DATA_BLOCK "DB_Z256_Scada"
{ DB_Accessible_From_OPC_UA := 'FALSE' ;
 DB_Accessible_From_Webserver := 'FALSE' ;
 S7_Optimized_Access := 'FALSE' }
VERSION : 0.1
NON_RETAIN
   STRUCT
      tAlm : Struct   // HMI Alarms
         tE { ExternalWritable := 'False'} : Struct
            x0 { ExternalWritable := 'False'} : Bool;   // KE.Main emergency on
            x1 { ExternalWritable := 'False'} : Bool;   // KE1.Local emergency on
            x2 { ExternalWritable := 'False'} : Bool;   // Cabinet.Emergency localization
            x3 { ExternalWritable := 'False'} : Bool;   // SB1.Emergency localization
            x4 { ExternalWritable := 'False'} : Bool;   // SB2.Emergency localization
            x5 { ExternalAccessible := 'False'; ExternalVisible := 'False'; ExternalWritable := 'False'} : Bool;
            x6 { ExternalAccessible := 'False'; ExternalVisible := 'False'; ExternalWritable := 'False'} : Bool;
            x7 { ExternalAccessible := 'False'; ExternalVisible := 'False'; ExternalWritable := 'False'} : Bool;
            x8 { ExternalAccessible := 'False'; ExternalVisible := 'False'; ExternalWritable := 'False'} : Bool;
            x9 { ExternalAccessible := 'False'; ExternalVisible := 'False'; ExternalWritable := 'False'} : Bool;
            x10 { ExternalAccessible := 'False'; ExternalVisible := 'False'; ExternalWritable := 'False'} : Bool;
            x11 { ExternalAccessible := 'False'; ExternalVisible := 'False'; ExternalWritable := 'False'} : Bool;
            x12 { ExternalAccessible := 'False'; ExternalVisible := 'False'; ExternalWritable := 'False'} : Bool;
            x13 { ExternalAccessible := 'False'; ExternalVisible := 'False'; ExternalWritable := 'False'} : Bool;
            x14 { ExternalAccessible := 'False'; ExternalVisible := 'False'; ExternalWritable := 'False'} : Bool;
            x15 { ExternalAccessible := 'False'; ExternalVisible := 'False'; ExternalWritable := 'False'} : Bool;
            x16 { ExternalAccessible := 'False'; ExternalVisible := 'False'; ExternalWritable := 'False'} : Bool;
            x17 { ExternalAccessible := 'False'; ExternalVisible := 'False'; ExternalWritable := 'False'} : Bool;
            x18 { ExternalAccessible := 'False'; ExternalVisible := 'False'; ExternalWritable := 'False'} : Bool;
            x19 { ExternalAccessible := 'False'; ExternalVisible := 'False'; ExternalWritable := 'False'} : Bool;
            x20 { ExternalAccessible := 'False'; ExternalVisible := 'False'; ExternalWritable := 'False'} : Bool;
            x21 { ExternalAccessible := 'False'; ExternalVisible := 'False'; ExternalWritable := 'False'} : Bool;
            x22 { ExternalAccessible := 'False'; ExternalVisible := 'False'; ExternalWritable := 'False'} : Bool;
            x23 { ExternalAccessible := 'False'; ExternalVisible := 'False'; ExternalWritable := 'False'} : Bool;
            x24 { ExternalAccessible := 'False'; ExternalVisible := 'False'; ExternalWritable := 'False'} : Bool;
            x25 { ExternalAccessible := 'False'; ExternalVisible := 'False'; ExternalWritable := 'False'} : Bool;
            x26 { ExternalAccessible := 'False'; ExternalVisible := 'False'; ExternalWritable := 'False'} : Bool;
            x27 { ExternalAccessible := 'False'; ExternalVisible := 'False'; ExternalWritable := 'False'} : Bool;
            x28 { ExternalAccessible := 'False'; ExternalVisible := 'False'; ExternalWritable := 'False'} : Bool;
            x29 { ExternalAccessible := 'False'; ExternalVisible := 'False'; ExternalWritable := 'False'} : Bool;
            x30 { ExternalAccessible := 'False'; ExternalVisible := 'False'; ExternalWritable := 'False'} : Bool;
            x31 { ExternalAccessible := 'False'; ExternalVisible := 'False'; ExternalWritable := 'False'} : Bool;
         END_STRUCT;
         tS { ExternalWritable := 'False'} : Struct
            tS0 { ExternalWritable := 'False'} : Struct
               x0 { ExternalWritable := 'False'} : Bool;   // xB18-3L+.PowerSupplyInputControlCabinetON
               x1 { ExternalWritable := 'False'} : Bool;   // xB18-7L+.InputInstallationPowerSupplyON"
               x2 { ExternalWritable := 'False'} : Bool;   // xB11QF1/1D/QF2.Anomaly power supplies 120V
               x3 { ExternalWritable := 'False'} : Bool;   // xB18QF2.Power supply 24V logic
               x4 { ExternalWritable := 'False'} : Bool;   // xB18QF3.Power supply 24V logic
               x5 { ExternalWritable := 'False'} : Bool;   // xB20QF2.Power supply 24V logic
               x6 { ExternalWritable := 'False'} : Bool;   // xB20QF3.Power supply 24V logic
               x7 { ExternalWritable := 'False'} : Bool;   // xB21QF1.Power supply 24V logic
               x8 { ExternalWritable := 'False'} : Bool;   // xB41QF1.ProtectionPowerSupplyMotorsYcut 1-4
               x9 { ExternalWritable := 'False'} : Bool;   // xB41QF2.Protection power supply 36V motors longitudinal cutting 1-4
               x10 { ExternalWritable := 'False'} : Bool;   // xB42QF1.ProtectionPowerSupplyMotorsYcut 5-8
               x11 { ExternalWritable := 'False'} : Bool;   // xB42QF2.Protection power supply 36V motors longitudinal cutting 5-8
               x12 { ExternalWritable := 'False'} : Bool;
               x13 { ExternalWritable := 'False'} : Bool;
               x14 { ExternalWritable := 'False'} : Bool;
               x15 { ExternalWritable := 'False'} : Bool;
               x16 { ExternalWritable := 'False'} : Bool;   // PLCA.Timeout receiving consumed message
               x17 { ExternalWritable := 'False'} : Bool;   // PLCB.Timeout receiving consumed message
               x18 { ExternalWritable := 'False'} : Bool;   // PLCA.Mission packet lost
               x19 { ExternalWritable := 'False'} : Bool;   // PLCB.Mission packet lost
               x20 { ExternalWritable := 'False'} : Bool;   // PLCA.Syncro packet lost
               x21 { ExternalWritable := 'False'} : Bool;   // PLCB.Syncro packet lost
               x22 { ExternalWritable := 'False'} : Bool;   // Syncro.YCut meter gap outside the limits
               x23 { ExternalWritable := 'False'} : Bool;   // Syncro.Main line meter gap outside the limits
               x24 { ExternalWritable := 'False'} : Bool;   // Syncro.Timeout receiving meter signal from main line
               x25 { ExternalWritable := 'False'} : Bool;   // Syncro.Timeout receiving syncro value from mainline
               x26 { ExternalWritable := 'False'} : Bool;   // Syncro.Unexpected syncro pulse
               x27 { ExternalWritable := 'False'} : Bool;   // Syncro.Unexpected syncro message
               x28 { ExternalWritable := 'False'} : Bool;   // Syncro.Machine not syncronized
               x29 { ExternalWritable := 'False'} : Bool;
               x30 { ExternalWritable := 'False'} : Bool;
               x31 { ExternalWritable := 'False'} : Bool;
            END_STRUCT;
            tS1 { ExternalWritable := 'False'} : Struct
               x0 { ExternalWritable := 'False'} : Bool;
               x1 { ExternalWritable := 'False'} : Bool;
               x2 { ExternalWritable := 'False'} : Bool;
               x3 { ExternalWritable := 'False'} : Bool;
               x4 { ExternalWritable := 'False'} : Bool;
               x5 { ExternalWritable := 'False'} : Bool;
               x6 { ExternalWritable := 'False'} : Bool;
               x7 { ExternalWritable := 'False'} : Bool;
               x8 { ExternalWritable := 'False'} : Bool;
               x9 { ExternalWritable := 'False'} : Bool;
               x10 { ExternalWritable := 'False'} : Bool;
               x11 { ExternalWritable := 'False'} : Bool;
               x12 { ExternalWritable := 'False'} : Bool;
               x13 { ExternalWritable := 'False'} : Bool;
               x14 { ExternalWritable := 'False'} : Bool;
               x15 { ExternalWritable := 'False'} : Bool;
               x16 { ExternalWritable := 'False'} : Bool;
               x17 { ExternalWritable := 'False'} : Bool;
               x18 { ExternalWritable := 'False'} : Bool;
               x19 { ExternalWritable := 'False'} : Bool;
               x20 { ExternalWritable := 'False'} : Bool;
               x21 { ExternalWritable := 'False'} : Bool;
               x22 { ExternalWritable := 'False'} : Bool;
               x23 { ExternalWritable := 'False'} : Bool;
               x24 { ExternalWritable := 'False'} : Bool;
               x25 { ExternalWritable := 'False'} : Bool;
               x26 { ExternalWritable := 'False'} : Bool;
               x27 { ExternalWritable := 'False'} : Bool;
               x28 { ExternalWritable := 'False'} : Bool;
               x29 { ExternalWritable := 'False'} : Bool;
               x30 { ExternalWritable := 'False'} : Bool;
               x31 { ExternalWritable := 'False'} : Bool;
            END_STRUCT;
            tS2 { ExternalWritable := 'False'} : Struct
               x0 { ExternalWritable := 'False'} : Bool;
               x1 { ExternalWritable := 'False'} : Bool;
               x2 { ExternalWritable := 'False'} : Bool;
               x3 { ExternalWritable := 'False'} : Bool;
               x4 { ExternalWritable := 'False'} : Bool;
               x5 { ExternalWritable := 'False'} : Bool;
               x6 { ExternalWritable := 'False'} : Bool;
               x7 { ExternalWritable := 'False'} : Bool;
               x8 { ExternalWritable := 'False'} : Bool;
               x9 { ExternalWritable := 'False'} : Bool;
               x10 { ExternalWritable := 'False'} : Bool;
               x11 { ExternalWritable := 'False'} : Bool;
               x12 { ExternalWritable := 'False'} : Bool;
               x13 { ExternalWritable := 'False'} : Bool;
               x14 { ExternalWritable := 'False'} : Bool;
               x15 { ExternalWritable := 'False'} : Bool;
               x16 { ExternalWritable := 'False'} : Bool;
               x17 { ExternalWritable := 'False'} : Bool;
               x18 { ExternalWritable := 'False'} : Bool;
               x19 { ExternalWritable := 'False'} : Bool;
               x20 { ExternalWritable := 'False'} : Bool;
               x21 { ExternalWritable := 'False'} : Bool;
               x22 { ExternalWritable := 'False'} : Bool;
               x23 { ExternalWritable := 'False'} : Bool;
               x24 { ExternalWritable := 'False'} : Bool;
               x25 { ExternalWritable := 'False'} : Bool;
               x26 { ExternalWritable := 'False'} : Bool;
               x27 { ExternalWritable := 'False'} : Bool;
               x28 { ExternalWritable := 'False'} : Bool;
               x29 { ExternalWritable := 'False'} : Bool;
               x30 { ExternalWritable := 'False'} : Bool;
               x31 { ExternalWritable := 'False'} : Bool;
            END_STRUCT;
            tS3 { ExternalWritable := 'False'} : Struct
               x0 { ExternalWritable := 'False'} : Bool;
               x1 { ExternalWritable := 'False'} : Bool;
               x2 { ExternalWritable := 'False'} : Bool;
               x3 { ExternalWritable := 'False'} : Bool;
               x4 { ExternalWritable := 'False'} : Bool;
               x5 { ExternalWritable := 'False'} : Bool;
               x6 { ExternalWritable := 'False'} : Bool;
               x7 { ExternalWritable := 'False'} : Bool;
               x8 { ExternalWritable := 'False'} : Bool;
               x9 { ExternalWritable := 'False'} : Bool;
               x10 { ExternalWritable := 'False'} : Bool;
               x11 { ExternalWritable := 'False'} : Bool;
               x12 { ExternalWritable := 'False'} : Bool;
               x13 { ExternalWritable := 'False'} : Bool;
               x14 { ExternalWritable := 'False'} : Bool;
               x15 { ExternalWritable := 'False'} : Bool;
               x16 { ExternalWritable := 'False'} : Bool;
               x17 { ExternalWritable := 'False'} : Bool;
               x18 { ExternalWritable := 'False'} : Bool;
               x19 { ExternalWritable := 'False'} : Bool;
               x20 { ExternalWritable := 'False'} : Bool;
               x21 { ExternalWritable := 'False'} : Bool;
               x22 { ExternalWritable := 'False'} : Bool;
               x23 { ExternalWritable := 'False'} : Bool;
               x24 { ExternalWritable := 'False'} : Bool;
               x25 { ExternalWritable := 'False'} : Bool;
               x26 { ExternalWritable := 'False'} : Bool;
               x27 { ExternalWritable := 'False'} : Bool;
               x28 { ExternalWritable := 'False'} : Bool;
               x29 { ExternalWritable := 'False'} : Bool;
               x30 { ExternalWritable := 'False'} : Bool;
               x31 { ExternalWritable := 'False'} : Bool;
            END_STRUCT;
         END_STRUCT;
         tF { ExternalAccessible := 'False'; ExternalVisible := 'False'; ExternalWritable := 'False'} : Struct
            x0 { ExternalAccessible := 'False'; ExternalVisible := 'False'; ExternalWritable := 'False'} : Bool;
            x1 { ExternalAccessible := 'False'; ExternalVisible := 'False'; ExternalWritable := 'False'} : Bool;
            x2 { ExternalAccessible := 'False'; ExternalVisible := 'False'; ExternalWritable := 'False'} : Bool;
            x3 { ExternalAccessible := 'False'; ExternalVisible := 'False'; ExternalWritable := 'False'} : Bool;
            x4 { ExternalAccessible := 'False'; ExternalVisible := 'False'; ExternalWritable := 'False'} : Bool;
            x5 { ExternalAccessible := 'False'; ExternalVisible := 'False'; ExternalWritable := 'False'} : Bool;
            x6 { ExternalAccessible := 'False'; ExternalVisible := 'False'; ExternalWritable := 'False'} : Bool;
            x7 { ExternalAccessible := 'False'; ExternalVisible := 'False'; ExternalWritable := 'False'} : Bool;
            x8 { ExternalAccessible := 'False'; ExternalVisible := 'False'; ExternalWritable := 'False'} : Bool;
            x9 { ExternalAccessible := 'False'; ExternalVisible := 'False'; ExternalWritable := 'False'} : Bool;
            x10 { ExternalAccessible := 'False'; ExternalVisible := 'False'; ExternalWritable := 'False'} : Bool;
            x11 { ExternalAccessible := 'False'; ExternalVisible := 'False'; ExternalWritable := 'False'} : Bool;
            x12 { ExternalAccessible := 'False'; ExternalVisible := 'False'; ExternalWritable := 'False'} : Bool;
            x13 { ExternalAccessible := 'False'; ExternalVisible := 'False'; ExternalWritable := 'False'} : Bool;
            x14 { ExternalAccessible := 'False'; ExternalVisible := 'False'; ExternalWritable := 'False'} : Bool;
            x15 { ExternalAccessible := 'False'; ExternalVisible := 'False'; ExternalWritable := 'False'} : Bool;
            x16 { ExternalAccessible := 'False'; ExternalVisible := 'False'; ExternalWritable := 'False'} : Bool;
            x17 { ExternalAccessible := 'False'; ExternalVisible := 'False'; ExternalWritable := 'False'} : Bool;
            x18 { ExternalAccessible := 'False'; ExternalVisible := 'False'; ExternalWritable := 'False'} : Bool;
            x19 { ExternalAccessible := 'False'; ExternalVisible := 'False'; ExternalWritable := 'False'} : Bool;
            x20 { ExternalAccessible := 'False'; ExternalVisible := 'False'; ExternalWritable := 'False'} : Bool;
            x21 { ExternalAccessible := 'False'; ExternalVisible := 'False'; ExternalWritable := 'False'} : Bool;
            x22 { ExternalAccessible := 'False'; ExternalVisible := 'False'; ExternalWritable := 'False'} : Bool;
            x23 { ExternalAccessible := 'False'; ExternalVisible := 'False'; ExternalWritable := 'False'} : Bool;
            x24 { ExternalAccessible := 'False'; ExternalVisible := 'False'; ExternalWritable := 'False'} : Bool;
            x25 { ExternalAccessible := 'False'; ExternalVisible := 'False'; ExternalWritable := 'False'} : Bool;
            x26 { ExternalAccessible := 'False'; ExternalVisible := 'False'; ExternalWritable := 'False'} : Bool;
            x27 { ExternalAccessible := 'False'; ExternalVisible := 'False'; ExternalWritable := 'False'} : Bool;
            x28 { ExternalAccessible := 'False'; ExternalVisible := 'False'; ExternalWritable := 'False'} : Bool;
            x29 { ExternalAccessible := 'False'; ExternalVisible := 'False'; ExternalWritable := 'False'} : Bool;
            x30 { ExternalAccessible := 'False'; ExternalVisible := 'False'; ExternalWritable := 'False'} : Bool;
            x31 { ExternalAccessible := 'False'; ExternalVisible := 'False'; ExternalWritable := 'False'} : Bool;
         END_STRUCT;
         tW { ExternalWritable := 'False'} : Struct
            x0 { ExternalWritable := 'False'} : Bool;   // PLCA.Timeout receiving consumed message
            x1 { ExternalWritable := 'False'} : Bool;   // PLCB.Timeout receiving consumed message
            x2 { ExternalWritable := 'False'} : Bool;   // PLCA.Mission packet lost
            x3 { ExternalWritable := 'False'} : Bool;   // PLCB.Mission packet lost
            x4 { ExternalWritable := 'False'} : Bool;   // PLCA.Syncro packet lost
            x5 { ExternalWritable := 'False'} : Bool;   // PLCB.Syncro packet lost
            x6 { ExternalWritable := 'False'} : Bool;   // QF.Protection air conditioners
            x7 { ExternalAccessible := 'False'; ExternalVisible := 'False'; ExternalWritable := 'False'} : Bool;
            x8 { ExternalAccessible := 'False'; ExternalVisible := 'False'; ExternalWritable := 'False'} : Bool;
            x9 { ExternalAccessible := 'False'; ExternalVisible := 'False'; ExternalWritable := 'False'} : Bool;
            x10 { ExternalAccessible := 'False'; ExternalVisible := 'False'; ExternalWritable := 'False'} : Bool;
            x11 { ExternalAccessible := 'False'; ExternalVisible := 'False'; ExternalWritable := 'False'} : Bool;
            x12 { ExternalAccessible := 'False'; ExternalVisible := 'False'; ExternalWritable := 'False'} : Bool;
            x13 { ExternalAccessible := 'False'; ExternalVisible := 'False'; ExternalWritable := 'False'} : Bool;
            x14 { ExternalAccessible := 'False'; ExternalVisible := 'False'; ExternalWritable := 'False'} : Bool;
            x15 { ExternalAccessible := 'False'; ExternalVisible := 'False'; ExternalWritable := 'False'} : Bool;
            x16 { ExternalAccessible := 'False'; ExternalVisible := 'False'; ExternalWritable := 'False'} : Bool;
            x17 { ExternalAccessible := 'False'; ExternalVisible := 'False'; ExternalWritable := 'False'} : Bool;
            x18 { ExternalAccessible := 'False'; ExternalVisible := 'False'; ExternalWritable := 'False'} : Bool;
            x19 { ExternalAccessible := 'False'; ExternalVisible := 'False'; ExternalWritable := 'False'} : Bool;
            x20 { ExternalAccessible := 'False'; ExternalVisible := 'False'; ExternalWritable := 'False'} : Bool;
            x21 { ExternalAccessible := 'False'; ExternalVisible := 'False'; ExternalWritable := 'False'} : Bool;
            x22 { ExternalAccessible := 'False'; ExternalVisible := 'False'; ExternalWritable := 'False'} : Bool;
            x23 { ExternalAccessible := 'False'; ExternalVisible := 'False'; ExternalWritable := 'False'} : Bool;
            x24 { ExternalAccessible := 'False'; ExternalVisible := 'False'; ExternalWritable := 'False'} : Bool;
            x25 { ExternalAccessible := 'False'; ExternalVisible := 'False'; ExternalWritable := 'False'} : Bool;
            x26 { ExternalAccessible := 'False'; ExternalVisible := 'False'; ExternalWritable := 'False'} : Bool;
            x27 { ExternalAccessible := 'False'; ExternalVisible := 'False'; ExternalWritable := 'False'} : Bool;
            x28 { ExternalAccessible := 'False'; ExternalVisible := 'False'; ExternalWritable := 'False'} : Bool;
            x29 { ExternalAccessible := 'False'; ExternalVisible := 'False'; ExternalWritable := 'False'} : Bool;
            x30 { ExternalAccessible := 'False'; ExternalVisible := 'False'; ExternalWritable := 'False'} : Bool;
            x31 { ExternalAccessible := 'False'; ExternalVisible := 'False'; ExternalWritable := 'False'} : Bool;
         END_STRUCT;
      END_STRUCT;
      tHMR { ExternalWritable := 'False'} : Struct   // HMI Read
         xCalibrationsAllowed { ExternalWritable := 'False'} : Bool;   // Calibration function allowed {x|x|x|x|O}
         xSpare1 { ExternalWritable := 'False'} : Bool;
         xSpare2 { ExternalWritable := 'False'} : Bool;
         xSpare3 { ExternalWritable := 'False'} : Bool;
         xSpare4 { ExternalWritable := 'False'} : Bool;
         xSpare5 { ExternalWritable := 'False'} : Bool;
         xSpare6 { ExternalWritable := 'False'} : Bool;
         xSpare7 { ExternalWritable := 'False'} : Bool;
         xSpare8 { ExternalWritable := 'False'} : Bool;
         xSpare9 { ExternalWritable := 'False'} : Bool;
         xSpare10 { ExternalWritable := 'False'} : Bool;
         xSpare11 { ExternalWritable := 'False'} : Bool;
         xSpare12 { ExternalWritable := 'False'} : Bool;
         xSpare13 { ExternalWritable := 'False'} : Bool;
         xSpare14 { ExternalWritable := 'False'} : Bool;
         xZoneAlarm { ExternalWritable := 'False'} : Bool;   // Zone alarm {X|X|X|X|O}
         xSpare16 { ExternalWritable := 'False'} : Bool;
         xSpare17 { ExternalWritable := 'False'} : Bool;
         xSpare18 { ExternalWritable := 'False'} : Bool;
         xSpare19 { ExternalWritable := 'False'} : Bool;
         xSpare20 { ExternalWritable := 'False'} : Bool;
         xSpare21 { ExternalWritable := 'False'} : Bool;
         xSpare22 { ExternalWritable := 'False'} : Bool;
         xSpare23 { ExternalWritable := 'False'} : Bool;
         xSpare24 { ExternalWritable := 'False'} : Bool;
         xSpare25 { ExternalWritable := 'False'} : Bool;
         xSpare26 { ExternalWritable := 'False'} : Bool;
         xSpare27 { ExternalWritable := 'False'} : Bool;
         xSpare28 { ExternalWritable := 'False'} : Bool;
         xSpare29 { ExternalWritable := 'False'} : Bool;
         xSpare30 { ExternalWritable := 'False'} : Bool;
         xSpare31 { ExternalWritable := 'False'} : Bool;
         xSpare { ExternalWritable := 'False'} : Array[0..15] of Bool;
         iSpare0 { ExternalWritable := 'False'} : Int;
         iSpare1 { ExternalWritable := 'False'} : Int;
         iSpare2 { ExternalWritable := 'False'} : Int;
         iSpare3 { ExternalWritable := 'False'} : Int;
         iSpare4 { ExternalWritable := 'False'} : Int;
         iSpare5 { ExternalWritable := 'False'} : Int;
         iSpare6 { ExternalWritable := 'False'} : Int;
         iSpare7 { ExternalWritable := 'False'} : Int;
         iSpare8 { ExternalWritable := 'False'} : Int;
         iSpare9 { ExternalWritable := 'False'} : Int;
         iSpare10 { ExternalWritable := 'False'} : Int;
         iSpare11 { ExternalWritable := 'False'} : Int;
         iSpare12 { ExternalWritable := 'False'} : Int;
         iSpare13 { ExternalWritable := 'False'} : Int;
         iSpare14 { ExternalWritable := 'False'} : Int;
         iSpare15 { ExternalWritable := 'False'} : Int;
         iSpare16 { ExternalWritable := 'False'} : Int;
         dZoneMode { ExternalWritable := 'False'} : DInt;   // Zone modality (1=Manual;4=Automatic;8=Manual request) {x|x|x|x|O}
         dZoneState { ExternalWritable := 'False'} : DInt;   // Zone status (1=CycleON 2=StopCyc 4=CycleReq 8=StopReq 1024=E-Stop) {X|X|X|X|O}
         dCabinetStatusMCC { ExternalWritable := 'False'} : DInt;   // Cabinet status MCC1256B (1=OK;2=General power alarm;3=Local power alarm) {X|X|X|X|O}
         dProdModeRequest { ExternalWritable := 'False'} : DInt;   // Production modality request (1=Out of Production 3= In production) {x|x|x|x|O}
         dProdModeActual { ExternalWritable := 'False'} : DInt;   // Production modality actual (1=Out of production 3=In production 8=Out of production request 9=In production request) {x|x|x|x|O}
         dSpare5 { ExternalWritable := 'False'} : DInt;
         "rgdHeadsActualStatus[0]" { ExternalWritable := 'False'} : DInt;   // Head #1 prod. status (1=Out of production 3=In production 8=Out of production request 9=In production request) {x|x|x|x|O}
         "rgdHeadsActualStatus[1]" { ExternalWritable := 'False'} : DInt;   // Head #2 prod. status (1=Out of production 3=In production 8=Out of production request 9=In production request) {x|x|x|x|O}
         "rgdHeadsActualStatus[2]" { ExternalWritable := 'False'} : DInt;   // Head #3 prod. status (1=Out of production 3=In production 8=Out of production request 9=In production request) {x|x|x|x|O}
         "rgdHeadsActualStatus[3]" { ExternalWritable := 'False'} : DInt;   // Head #4 prod. status (1=Out of production 3=In production 8=Out of production request 9=In production request) {x|x|x|x|O}
         "rgdHeadsActualStatus[4]" { ExternalWritable := 'False'} : DInt;   // Head #5 prod. status (1=Out of production 3=In production 8=Out of production request 9=In production request) {x|x|x|x|O}
         "rgdHeadsActualStatus[5]" { ExternalWritable := 'False'} : DInt;   // Head #6 prod. status (1=Out of production 3=In production 8=Out of production request 9=In production request) {x|x|x|x|O}
         "rgdHeadsActualStatus[6]" { ExternalWritable := 'False'} : DInt;   // Head #7 prod. status (1=Out of production 3=In production 8=Out of production request 9=In production request) {x|x|x|x|O}
         "rgdHeadsActualStatus[7]" { ExternalWritable := 'False'} : DInt;   // Head #8 prod. status (1=Out of production 3=In production 8=Out of production request 9=In production request) {x|x|x|x|O}
         dSpare14 { ExternalWritable := 'False'} : DInt;
         dSpare15 { ExternalWritable := 'False'} : DInt;
         dSpare { ExternalWritable := 'False'} : Array[0..15] of DInt;
         rSpare0 { ExternalWritable := 'False'} : Real;
         rSpare1 { ExternalWritable := 'False'} : Real;
         rSpare2 { ExternalWritable := 'False'} : Real;
         rSpare3 { ExternalWritable := 'False'} : Real;
         rSpare4 { ExternalWritable := 'False'} : Real;
         rSpare5 { ExternalWritable := 'False'} : Real;
         rSpare6 { ExternalWritable := 'False'} : Real;
         rSpare7 { ExternalWritable := 'False'} : Real;
         rSpare8 { ExternalWritable := 'False'} : Real;
         tManCmd { ExternalWritable := 'False'} : Struct
            xSpare0 { ExternalWritable := 'False'} : Bool;
            xSpare1 { ExternalWritable := 'False'} : Bool;
            xSpare2 { ExternalWritable := 'False'} : Bool;
            xSpare3 { ExternalWritable := 'False'} : Bool;
            xSpare4 { ExternalWritable := 'False'} : Bool;
            xSpare5 { ExternalWritable := 'False'} : Bool;
            xSpare6 { ExternalWritable := 'False'} : Bool;
            xSpare7 { ExternalWritable := 'False'} : Bool;
            xSpare8 { ExternalWritable := 'False'} : Bool;
            xSpare9 { ExternalWritable := 'False'} : Bool;
            xSpare10 { ExternalWritable := 'False'} : Bool;
            xSpare11 { ExternalWritable := 'False'} : Bool;
            xSpare12 { ExternalWritable := 'False'} : Bool;
            xSpare13 { ExternalWritable := 'False'} : Bool;
            xSpare14 { ExternalWritable := 'False'} : Bool;
            xSpare15 { ExternalWritable := 'False'} : Bool;
            xSpare { ExternalWritable := 'False'} : Array[0..15] of Bool;
         END_STRUCT;
      END_STRUCT;
      tHMW : Struct   // HMI Write
         xAutoModeReq : Bool;   // Automatic mode request {x|x|x|x|O}
         xManModeReq : Bool;   // Manual mode request {x|x|x|x|O}
         xOutOfProdReq : Bool;   // Bridge out of production request {x|x|x|x|O}
         xInProdReq : Bool;   // Bridge in production request {x|x|x|x|O}
         xCutOnBreakEnabled { ExternalWritable := 'False'} : Bool;   // Cut during glass break {x|x|x|x|O}
         xMotorsAndCardsInitialize : Bool;   // Motors and cards initialize {x|x|x|x|M}
         xForceHeadsHoming : Bool;   // Force the homing of the heads {x|x|x|x|M}
         xPositionCalibrationRequest : Bool;   // Position calibration request {x|x|x|x|M}
         xBridgeOffsetCalibrationRequest : Bool;   // Bridge offset calibration request {x|x|x|x|M}
         xSpare9 { ExternalWritable := 'False'} : Bool;   //
         xSpare10 : Bool;   //
         xSpare11 : Bool;   //
         xSpare12 : Bool;
         xSpare13 : Bool;
         xGeneralReset : Bool;   // General reset {X|X|X|X|M}
         xFaultsReset : Bool;   // Reset faults {X|X|X|X|O}
         xHeadEnabled_1 { ExternalWritable := 'False'} : Bool;   // Head #1 enabled/disabled {x|x|x|x|O}
         xHeadEnabled_2 { ExternalWritable := 'False'} : Bool;   // Head #2 enabled/disabled {x|x|x|x|O}
         xHeadEnabled_3 { ExternalWritable := 'False'} : Bool;   // Head #3 enabled/disabled {x|x|x|x|O}
         xHeadEnabled_4 { ExternalWritable := 'False'} : Bool;   // Head #4 enabled/disabled {x|x|x|x|O}
         xHeadEnabled_5 { ExternalWritable := 'False'} : Bool;   // Head #5 enabled/disabled {x|x|x|x|O}
         xHeadEnabled_6 { ExternalWritable := 'False'} : Bool;   // Head #6 enabled/disabled {x|x|x|x|O}
         xHeadEnabled_7 { ExternalWritable := 'False'} : Bool;   // Head #7 enabled/disabled {x|x|x|x|O}
         xHeadEnabled_8 { ExternalWritable := 'False'} : Bool;   // Head #8 enabled/disabled {x|x|x|x|O}
         xSpare24 : Bool;
         xSpare25 : Bool;
         xSpare26 : Bool;
         xSpare27 : Bool;
         xSpare28 : Bool;
         xSpare29 : Bool;
         xSpare30 : Bool;
         xSpare31 : Bool;
         xSpare : Array[0..15] of Bool;
         iSpare0 : Int;
         iSpare1 : Int;
         iSpare2 : Int;
         iSpare3 : Int;
         iSpare4 : Int;
         iSpare5 : Int;
         iSpare6 : Int;
         iSpare7 : Int;
         iSpare8 : Int;
         iSpare9 : Int;
         iSpare10 : Int;
         iSpare11 : Int;
         iSpare12 : Int;
         iSpare13 : Int;
         iSpare14 : Int;
         iSpare15 : Int;
         iSpare16 : Int;
         dNumberOfLites : DInt;   // Calibration. number of lite on calibration {x|x|1|8|M}
         dMoveBridgeOffset_cmm : DInt;   // Calibration. Move all the heads of this offset {mm/100|mm|-100|100|M}
         dPressureScalerOnSample_perc : DInt;   // Pressure scaler during sample plate [%] {%|%|0|100|O}
         dSpare3 : DInt;
         dSpare4 : DInt;
         dSpare5 : DInt;
         dSpare6 : DInt;
         dSpare7 : DInt;
         dHead_Selected_1 : DInt;   // Calibration. head number selected Cut1 {x|x|1|11|M}
         dHead_Selected_2 : DInt;   // Calibration. head number selected Cut2 {x|x|1|11|M}
         dHead_Selected_3 : DInt;   // Calibration. head number selected Cut3{x|x|1|11|M}
         dHead_Selected_4 : DInt;   // Calibration. head number selected Cut4{x|x|1|11|M}
         dHead_Selected_5 : DInt;   // Calibration. head number selected Cut5{x|x|1|11|M}
         dHead_Selected_6 : DInt;   // Calibration. head number selected Cut6{x|x|1|11|M}
         dHead_Selected_7 : DInt;   // Calibration. head number selected Cut7{x|x|1|11|M}
         dHead_Selected_8 : DInt;   // Calibration. head number selected Cut8{x|x|1|11|M}
         dCutWidthTeo_cmm_1 : DInt;   // Calibration. cut width Lite 1 theorical [mm/100] {mm/100|mm|200|4000|M}
         dCutWidthTeo_cmm_2 : DInt;   // Calibration. cut width Lite 2 theorical [mm/100] {mm/100|mm|200|4000|M}
         dCutWidthTeo_cmm_3 : DInt;   // Calibration. cut width Lite 3 theorical [mm/100] {mm/100|mm|200|4000|M}
         dCutWidthTeo_cmm_4 : DInt;   // Calibration. cut width Lite 4 theorical [mm/100] {mm/100|mm|200|4000|M}
         dCutWidthTeo_cmm_5 : DInt;   // Calibration. cut width Lite 5 theorical [mm/100] {mm/100|mm|200|4000|M}
         dCutWidthTeo_cmm_6 : DInt;   // Calibration. cut width Lite 6 theorical [mm/100] {mm/100|mm|200|4000|M}
         dCutWidthTeo_cmm_7 : DInt;   // Calibration. cut width Lite 7 theorical [mm/100] {mm/100|mm|200|4000|M}
         dCutWidthTeo_cmm_8 : DInt;   // Calibration. cut width Lite 8 theorical [mm/100] {mm/100|mm|200|4000|M}
         dCutWidthReal_cmm_1 : DInt;   // Calibration. cut width Lite 1 real [mm/100] {mm/100|mm|200|4000|M}
         dCutWidthReal_cmm_2 : DInt;   // Calibration. cut width Lite 2 real [mm/100] {mm/100|mm|200|4000|M}
         dCutWidthReal_cmm_3 : DInt;   // Calibration. cut width Lite 3 real [mm/100] {mm/100|mm|200|4000|M}
         dCutWidthReal_cmm_4 : DInt;   // Calibration. cut width Lite 4 real [mm/100] {mm/100|mm|200|4000|M}
         dCutWidthReal_cmm_5 : DInt;   // Calibration. cut width Lite 5 real [mm/100] {mm/100|mm|200|4000|M}
         dCutWidthReal_cmm_6 : DInt;   // Calibration. cut width Lite 6 real [mm/100] {mm/100|mm|200|4000|M}
         dCutWidthReal_cmm_7 : DInt;   // Calibration. cut width Lite 7 real [mm/100] {mm/100|mm|200|4000|M}
         dCutWidthReal_cmm_8 : DInt;   // Calibration. cut width Lite 8 real [mm/100] {mm/100|mm|200|4000|M}
         dSpare32 : DInt;
         dSpare33 : DInt;
         dSpare34 : DInt;
         dSpare35 : DInt;
         dSpare36 : DInt;
         dSpare37 : DInt;
         dSpare38 : DInt;
         dSpare39 : DInt;
         dSpare { ExternalWritable := 'False'} : Array[0..19] of DInt;
         rSpare0 : Real;
         rSpare1 : Real;
         rSpare2 : Real;
         rSpare3 : Real;
         rSpare4 : Real;
         rSpare5 : Real;
         rSpare6 : Real;
         rSpare7 : Real;
         rSpare8 : Real;
         tManCmd : Struct
            xBrakeEngage : Bool;   // Brake engage all heads {x|x|x|x|O}
            xBrakeRelease : Bool;   // Brake release all heads {x|x|x|x|O}
            xSpare2 { ExternalWritable := 'False'} : Bool;
            xSpare3 { ExternalWritable := 'False'} : Bool;
            xSpare4 { ExternalWritable := 'False'} : Bool;
            xSpare5 { ExternalWritable := 'False'} : Bool;
            xSpare6 { ExternalWritable := 'False'} : Bool;
            xSpare7 { ExternalWritable := 'False'} : Bool;
            xSpare8 { ExternalWritable := 'False'} : Bool;
            xSpare9 { ExternalWritable := 'False'} : Bool;
            xSpare10 { ExternalWritable := 'False'} : Bool;
            xSpare11 { ExternalWritable := 'False'} : Bool;
            xSpare12 { ExternalWritable := 'False'} : Bool;
            xSpare13 { ExternalWritable := 'False'} : Bool;
            xSpare14 { ExternalWritable := 'False'} : Bool;
            xSpare15 { ExternalWritable := 'False'} : Bool;
            xSpare16 : Bool;
            xSpare17 : Bool;
            xSpare18 : Bool;
            xSpare19 : Bool;
            xSpare20 : Bool;
            xSpare21 : Bool;
            xSpare22 : Bool;
            xSpare23 : Bool;
            xSpare24 : Bool;
            xSpare25 : Bool;
            xSpare26 : Bool;
            xSpare27 : Bool;
            xSpare28 : Bool;
            xSpare29 : Bool;
            xSpare30 : Bool;
            xSpare31 : Bool;
         END_STRUCT;
      END_STRUCT;
   END_STRUCT;


BEGIN
   tHMR.xCalibrationsAllowed := FALSE;
   tHMR.xZoneAlarm := FALSE;
   tHMR.dZoneMode := 4;
   tHMR.dZoneState := 1024;
   tHMR.dCabinetStatusMCC := 1;
   tHMR.dProdModeRequest := 3;
   tHMR.dProdModeActual := 3;
   tHMR."rgdHeadsActualStatus[0]" := 3;
   tHMR."rgdHeadsActualStatus[1]" := 3;
   tHMR."rgdHeadsActualStatus[2]" := 3;
   tHMR."rgdHeadsActualStatus[3]" := 3;
   tHMW.xAutoModeReq := FALSE;
   tHMW.xManModeReq := FALSE;
   tHMW.xOutOfProdReq := FALSE;
   tHMW.xInProdReq := FALSE;
   tHMW.xCutOnBreakEnabled := FALSE;
   tHMW.xMotorsAndCardsInitialize := FALSE;
   tHMW.xForceHeadsHoming := FALSE;
   tHMW.xPositionCalibrationRequest := FALSE;
   tHMW.xBridgeOffsetCalibrationRequest := FALSE;
   tHMW.xGeneralReset := FALSE;
   tHMW.xFaultsReset := FALSE;
   tHMW.xHeadEnabled_1 := TRUE;
   tHMW.xHeadEnabled_2 := TRUE;
   tHMW.xHeadEnabled_3 := TRUE;
   tHMW.xHeadEnabled_4 := TRUE;
   tHMW.xHeadEnabled_5 := TRUE;
   tHMW.xHeadEnabled_6 := TRUE;
   tHMW.xHeadEnabled_7 := TRUE;
   tHMW.xHeadEnabled_8 := TRUE;
   tHMW.dNumberOfLites := 1;
   tHMW.dMoveBridgeOffset_cmm := 0;
   tHMW.dPressureScalerOnSample_perc := 100;
   tHMW.tManCmd.xBrakeEngage := FALSE;
   tHMW.tManCmd.xBrakeRelease := FALSE;

END_DATA_BLOCK

